TYPE ST_PB_SG_InputsCommand :
(**************************************************************************************
 * 	Application		:	BoxControl Framework
 *	Revision		:	$Revision: 417092 $
 *	Revision date	:	$Date: 2018-11-14 12:58:58 +0100 (Mi., 14 Nov 2018) $
 *	Last changed by	:	$Author: q8aberh $
 *	URL				:	$URL: http://almscdc.swisslog.com/repo/SWPD/Development/ProMove/02_Controls/ProBox/03_Implementation/01_DevelopmentProject/01_Software/ProBox_COE/ProBox_DevProj_v1.0/PLC_1/20_Product/10_App/14_Groups/10_Lib/10_Conv/01_DUTs/10_Dummy/ST_SG_InputsCommand.T $
 *
 *	Purpose			:	Switching group inputs - commands.
 *
 * ------------------------------------------------------------------------------------
 *	Copyright Swisslog [IP AG], Switzerland. All rights reserved.
 * 
 * ------------------------------------------------------------------------------------
 *	
 * 	Revision History: 
 *
 * 	VERSION			DATE			INITIALS			DESCRIPTION
 *	0.1				01.01.2001		swl					Example
 *
 **************************************************************************************)
STRUCT
	AutoMode				: BOOL;	// Auto mode
	ManualMode				: BOOL; // Manual mode
	SemiAutoMode			: BOOL; // Semi auto mode
	StartPB					: BOOL;	// Start push button
	StopPB					: BOOL; // Stop push button
	StartStopPB				: BOOL; // Start stop push button
	ResetErrorPB			: BOOL; // Reset Error push button
	ResetEmgPB				: BOOL; // Reset Emg push button	
	
	
END_STRUCT
END_TYPE

(* stored: Version 1.1.0.1, ProductVersion 3.1.4024.9
   DUT ST_PB_SG_InputsCommand: Id {a32ac111-9c88-4868-9f94-acc21e19d45e} *)
